(* IEC 61131-3 sources: iec-checker/test/st/good, 22 files *)

(* ---- function-declaration.st ---- *)
(* Test for declaration of Function POU. *)
FUNCTION fn1 : INT
    VAR_INPUT
        vi1 : INT;
        vi2 : DINT;
    END_VAR
    VAR_OUTPUT
        vo1 : INT;
    END_VAR
    VAR_IN_OUT
        vio1 : INT;
    END_VAR
    VAR_IN_OUT
        vio1 : INT;
    END_VAR
    VAR
        v1 : INT;
    END_VAR
    VAR_EXTERNAL
        ve1 : INT;
    END_VAR
    VAR_TEMP
        vt1 : INT;
    END_VAR

    vio1 := 42;
END_FUNCTION

(* ---- generic-types.st ---- *)
(* Extended example from Beckhoff: https://infosys.beckhoff.com/english.php?content=../content/1033/tc3_plc_intro/18014401038986379.html&id= *)
FUNCTION F_AnyBitFunc : BOOL
VAR_INPUT
  value : ANY_BIT;
END_VAR
  value := 0;
END_FUNCTION

FUNCTION F_AnyDateFunc : BOOL
VAR_INPUT
    value : ANY_DATE;
END_VAR
  value := 0;
END_FUNCTION

FUNCTION F_AnyFunc : BOOL
VAR_INPUT
    value : ANY;
END_VAR
  value := 0;
END_FUNCTION

FUNCTION F_AnyIntFunc : BOOL
VAR_INPUT
    value : ANY_INT;
END_VAR
  value := 0;
END_FUNCTION

FUNCTION F_AnyNumFunc : BOOL
VAR_INPUT
    value : ANY_NUM;
END_VAR
  value := 0;
END_FUNCTION

FUNCTION F_AnyRealFunc : BOOL
VAR_INPUT
    value : ANY_REAL;
END_VAR
  value := 0;
END_FUNCTION

FUNCTION F_AnyStringFunc : BOOL
VAR_INPUT
    value : ANY_STRING;
END_VAR
  value := 0;
END_FUNCTION

(* ---- array-use.st ---- *)
FUNCTION_BLOCK MAIN_POU

  VAR
      i:INT;
      state: INT:=0;
  END_VAR

   IF gvl.CALL_LIST_INTERMEDIATE_GO_UP[i]= TRUE THEN
      state:=100;
  END_IF

END_FUNCTION_BLOCK

(* ---- empty-body.st ---- *)
(* Allow POU that contains only {} in their bodies. *)
FUNCTION EmptyFun : BOOL
  {}
END_FUNCTION

FUNCTION_BLOCK EmptyFB
  {}
END_FUNCTION_BLOCK

PROGRAM EmptyProgram
  {}
END_PROGRAM

(* ---- function-blocks.st ---- *)
FUNCTION_BLOCK fb0
END_FUNCTION_BLOCK

FUNCTION_BLOCK fb1
  VAR_INPUT
    vi1 : DINT;
  END_VAR
  VAR_OUTPUT
    vo1 : DINT;
  END_VAR
  VAR_IN_OUT
    vio1 : DINT;
  END_VAR
  VAR
    v1 : DINT;
  END_VAR
  VAR_TEMP
    vt1 : DINT;
  END_VAR
  VAR RETAIN
    vr1 : DINT;
  END_VAR
  VAR NON_RETAIN
    vnr1 : DINT;
  END_VAR
  v1 := 42;
END_FUNCTION_BLOCK

(* ---- references.st ---- *)
FUNCTION_BLOCK fb1
  VAR_INPUT
    vi1 : DINT;
  END_VAR
  v1 := 42;
END_FUNCTION_BLOCK

PROGRAM example
  VAR
    temp : DINT;
  END_VAR

  temp ?= temp^;
  temp ?= temp^^;
  temp ?= temp^^^;
  temp ?= NULL;
  temp ?= fb1;
END_PROGRAM

(* ---- simple.st ---- *)
FUNCTION_BLOCK Example
    VAR_EXTERNAL
        global_var : INT;
    END_VAR
    global_var := 42;
END_FUNCTION_BLOCK

PROGRAM Simple
  VAR_INPUT
    x : TIME;
  END_VAR
  VAR
    temp : DINT;
    i : DINT;
    arr1: ARRAY [1..2] OF BOOL;
    unused_var AT %IW1.2 : REAL := 200.0;
    head AT %B0 : INT;
  END_VAR

  WHILE i < 10 DO
    IF i = 5 THEN
      temp := i;
      EXIT;
      i := 42;
    END_IF
    i := i + 1;
  END_WHILE

  ARR1[3] := 19;
  ARR1[2,1] := 19;
  IF x = T#100MS THEN
    %B0 := 42;
  END_IF
END_PROGRAM

(* ---- user3.st ---- *)
FUNCTION_BLOCK MAIN_POU

  VAR_INPUT
  END_VAR

  VAR_OUTPUT
  END_VAR

  VAR
      FB4_Populate_Intermediate_Call_List_call : FB4_Populate_Intermediate_Call_List;
      FB5_Trigger_FB2_Call_FIFO_call:FB5_Trigger_FB2_Call_FIFO;
      MC_power_X1 : MC_Power;
      MC_readAxisPosition_jog:MC_ReadActualPosition;
      MC_ReadStatus_jog:MC_ReadStatus;
      MC_jog:MC_Jog;
      MC_Halt_jog:MC_Halt;
      MC_Stop_jog:MC_Stop;
      MC_Reset_jog:MC_Reset;
      MC_MoveAbsolute_jog:MC_MoveAbsolute;
      mainMotor:Motor;
      ton_0 : TON;
      ton_1 : TON;
      ton_2 : TON;
      axisPosition:REAL;
      nextTargetFloor:INT;
      nextTargetPosition:REAL;
      nextIntermediateTargetPosition:REAL;
      nextIntermediateTargetFloor:INT;
      nextIntermediateTargetFloorAvailable:bool;
      lastTargetFloor:INT;
      currentFloorNumber_:INT;
      i:INT;
      state: INT:=0;
      test_READ:BOOL;
      test_FORWARD:BOOL;
  END_VAR

  // Write values to Global Variables
  gvl.state_POU_1:=state;
  gvl.QW_axisPosition:=axisPosition;

  // Read axis position all the time
  MC_readAxisPosition_jog(Axis:=X1,
      Enable:=TRUE,
      Position=>axisPosition);

  // Motor Halt
  IF mainMotor.IX_Halt THEN
      MC_jog(Axis:=X1,
          JogForward:=FALSE,
          JogBackward:=FALSE);
  END_IF

  // Main Power
  mainMotor.IX_Power:=TRUE;
  IF mainMotor.IX_Power THEN
      MC_power_X1(Axis:=X1,
          Enable:=TRUE,
          bRegulatorOn:=TRUE,
          bDriveStart:=TRUE);
  ELSE
      MC_power_X1(Axis:=X1,
          Enable:=FALSE,
          bRegulatorOn:=FALSE,
          bDriveStart:=FALSE);
  END_IF

  // STOP/RESET the motor
  MC_Stop_jog(Axis:=X1,
      Execute:=mainMotor.IX_Stop,
      Deceleration:=5);
  MC_Reset_jog(Axis:=X1,
      Execute:=mainMotor.IX_Reset);

  // Drive error ID
  gvl.jogErrorID := MC_jog.ErrorId;

  CASE state OF
      0:  // Power ON
          IF MC_power_X1.Status = TRUE THEN
              ton_0(IN:=NOT ton_0.Q,PT:=1);
              IF ton_0.Q THEN
                  state := 10;
              END_IF
          END_IF

      10:
          IF nextIntermediateTargetFloorAvailable=FALSE THEN
              FB5_Trigger_FB2_Call_FIFO_call(POP:=2);
              IF FB5_Trigger_FB2_Call_FIFO_call.done = TRUE THEN
                  state:=11;
              END_IF
          ELSE
              state:=11;
          END_IF

      11:
          IF gvl.Dout <>0 THEN
              state:=12;
          ELSE
              state:=10;
          END_IF

      12:
          gvl.targetPosition := WORD_TO_INT(gvl.Dout-1)*gvl.floor_to_floor_distance;
          nextTargetFloor := WORD_TO_INT(gvl.Dout);

          IF gvl.Dout <> 0 AND gvl.targetPosition <> gvl.QW_axisPosition THEN
              IF gvl.QW_axisPosition < gvl.targetPosition THEN
                  gvl.jogDirection:='GO_UP';
                  MC_jog(Axis:=X1,
                          JogForward:=TRUE,
                          Velocity:=gvl.velocity_high,
                          Acceleration:=gvl.acceleration_high,
                          Deceleration:=gvl.deceleration_high);
              ELSIF gvl.QW_axisPosition > gvl.targetPosition THEN
                  gvl.jogDirection:='GO_DOWN';
                  MC_jog(Axis:=X1,
                          JogBackward:=TRUE,
                          Velocity:=gvl.velocity_high,
                          Acceleration:=gvl.acceleration_high,
                          Deceleration:=gvl.deceleration_high);
              END_IF
          ELSE
              state:=10;
          END_IF

          FB4_Populate_Intermediate_Call_List_call();
          IF gvl.jogDirection='GO_UP' THEN
              // If intermediate floor calls available_GO_UP
              FOR i:=1 TO gvl.NUM_FLOOR DO
                   IF gvl.CALL_LIST_INTERMEDIATE_GO_UP[i]= TRUE AND gvl.QW_axisPosition > (i-1)*gvl.floor_to_floor_distance-200 THEN
                      MC_jog(Axis:=X1,
                          JogForward:=FALSE,
                          JogBackward:=FALSE);
                      nextIntermediateTargetFloor:=i;
                      gvl.nextIntermediateTargetPosition:=(i-1)*gvl.floor_to_floor_distance;
                      state:=100;
                  END_IF
              END_FOR
              // If NO intermediate floor calls available
              IF gvl.QW_axisPosition > gvl.targetPosition-400 THEN
                  MC_jog(Axis:=X1,
                  JogForward:=FALSE,
                  JogBackward:=FALSE);
              END_IF
              IF MC_jog.Busy=FALSE THEN
                  state:=102;
              END_IF
          END_IF

          IF gvl.jogDirection='GO_DOWN' THEN
              // If intermediate floor calls available_GO_DOWN
              FOR i:=1 TO gvl.NUM_FLOOR DO
                   IF gvl.CALL_LIST_INTERMEDIATE_GO_DOWN[i]= TRUE AND gvl.QW_axisPosition < (i-1)*gvl.floor_to_floor_distance+200 THEN
                      MC_jog(Axis:=X1,
                          JogForward:=FALSE,
                          JogBackward:=FALSE);
                      nextIntermediateTargetFloor:=i;
                      gvl.nextIntermediateTargetPosition:=(i-1)*gvl.floor_to_floor_distance;
                      state:=100;
                  END_IF
              END_FOR
              // If NO intermediate floor calls available
              IF gvl.QW_axisPosition < gvl.targetPosition+400 THEN
                  MC_jog(Axis:=X1,
                  JogForward:=FALSE,
                  JogBackward:=FALSE);
              END_IF
              IF MC_jog.Busy=FALSE THEN
                  state:=102;
              END_IF
          END_IF

      100: // If YES intermediate floor calls available
          MC_MoveAbsolute_jog(Axis:=X1,
              Execute:=TRUE,
              Position:=gvl.nextIntermediateTargetPosition,
              Velocity:=gvl.velocity_low,
              Acceleration:=gvl.acceleration_low,
              Deceleration:=gvl.deceleration_low);

          IF MC_MoveAbsolute_jog.Done THEN
              MC_MoveAbsolute_jog(Axis:=X1,
                  Execute:=FALSE);
              nextIntermediateTargetFloorAvailable:=TRUE;
              state:=400;
          END_IF;

      102: // If NO intermediate floor calls available
          MC_MoveAbsolute_jog(Axis:=X1,
              Execute:=TRUE,
              Position:=gvl.targetPosition,
              Velocity:=gvl.velocity_low,
              Acceleration:=gvl.acceleration_low,
              Deceleration:=gvl.deceleration_low);

          IF MC_MoveAbsolute_jog.Done THEN
              MC_MoveAbsolute_jog(Axis:=X1,
                  Execute:=FALSE);
              nextIntermediateTargetFloorAvailable:=FALSE;
              state:=400;
          END_IF

      400: // Door closed and all safety OK.
          currentFloorNumber_:=FC1_currentFloorNumber(axisPosition:=axisPosition);
          gvl.Din_toRemove := INT_TO_WORD(currentFloorNumber_);

          gvl.CALL_LIST[currentFloorNumber_]:=FALSE;
          gvl.CALL_LIST_INTERMEDIATE_GO_DOWN[currentFloorNumber_]:=FALSE;
          gvl.CALL_LIST_INTERMEDIATE_GO_UP[currentFloorNumber_]:=FALSE;

          FB5_Trigger_FB2_Call_FIFO_call(POP:=3);
          IF FB5_Trigger_FB2_Call_FIFO_call.done = TRUE THEN
              state:=402;
          END_IF

      402:
          IF GVL.IX_DoorClosedAndAllSafetyOk THEN
              state:=10;
          END_IF

  END_CASE

END_FUNCTION_BLOCK

(* ---- array-in-loop.st ---- *)
PROGRAM Simple

  VAR
    i : DINT;
    arr1: ARRAY [1..2] OF BOOL;
  END_VAR

  VAR
    unused_var AT %IW1.2 : REAL := 200.0;
  END_VAR

  IF ARR1[i] < 10 THEN
    i := i + 1;
  END_IF;
END_PROGRAM

(* ---- case-insensitive.st ---- *)
(* Keywords and identifiers are case-insensitive *)
Program simple
  VaR
    v01 : DiNt;
  eND_var

  v01 := 92;
  V01 := 92;
END_PROGRAM

PRoGRAM square_root
  var
    a, b, c, d : REAL;
    x1, x2 : REaL;
    nroots : InT;
  END_VAR

  d := b*b - 4.0*a;
  d := b*b - 4.0*a*c;
  IF d < 0.0
  THEN nroots := 0;
    ELSIF d = 0.0
    THEN
      nroots := 1;
      X1 := -b/(2.0*A);
      X1 := -b;
    ELSE
      nroots := 2;
      X1 := (-b + SQRT(d))/(2.0*a);
      X2 := (-b - SQRT(d))/(2.0*a);
  END_IF;

ENd_ProGRAM

(* ---- comments.st ---- *)
PROGRAM comments
	VAR
		INITIAL : BOOL := FALSE;
		X1 : INT := 10;
		Y1 : INT := 20;
    // Test
	END_VAR
  // Test1
	Y1 := Z + 1; // Test2
	O_I1 := Y1; // Test3
END_PROGRAM

(* ---- configurations.st ---- *)
(* Demo program with all possible TASK entries.
   Created with Beremiz IDE (https://beremiz.org/). *)
FUNCTION function0 : BOOL
  VAR
    LocalVar0 : DINT;
  END_VAR

  LocalVar0 := 42;
END_FUNCTION

PROGRAM program0
  VAR
    LocalVar0 : DINT;
    LocalVar1 : TOD;
  END_VAR

  LocalVar0 := 42;
END_PROGRAM

PROGRAM program1
  VAR
    LocalVar0 : DINT;
  END_VAR

  LocalVar0 := 16#42;
END_PROGRAM

CONFIGURATION config
  VAR_GLOBAL
    ConfVar0 : DINT;
    ConfVar1 : DINT;
    ConfVar2 : DINT;
  END_VAR

  RESOURCE resource1 ON PLC
    VAR_GLOBAL
      ResVar0 : DINT;
      ResVar1 : BOOL;
    END_VAR
    TASK task0(INTERVAL := T#20ms,PRIORITY := 0);
    TASK task1(SINGLE := ResVar1,PRIORITY := 0);
    TASK task2(INTERVAL := T#2h0m0s3ms,PRIORITY := 1);
    PROGRAM instance0 WITH task0 : program0;
    PROGRAM instance1 WITH task1 : program1;
    PROGRAM instance2 WITH task2 : program1;
  END_RESOURCE
END_CONFIGURATION

(* ---- control-statements.st ---- *)
(* This file contains various control statements of the ST language. *)

(* Table 72 -- №4 *)
PROGRAM square_root
  VAR
    a, b, c, d : REAL;
    x1, x2 : REAL;
    nroots : INT;
  END_VAR

  d := b*b - 4.0*a;
  d := b*b - 4.0*a*c;
  IF d < 0.0
  THEN nroots := 0;
    ELSIF d = 0.0
    THEN
      nroots := 1;
      X1 := -b/(2.0*A);
      X1 := -b;
    ELSE
      nroots := 2;
      X1 := (-b + SQRT(d))/(2.0*a);
      X2 := (-b - SQRT(d))/(2.0*a);
  END_IF;

END_PROGRAM

PROGRAM test_for
  VAR
    i, j : INT;
    flag : INT;
    counter : INT := 0;
    some_var : INT;
  END_VAR

  FOR i := 0 TO 10 DO
    FOR j := 10 TO 100 BY 2 DO
      IF flag THEN
        EXIT;
      END_IF;
      counter := counter + 1;
      IF j = 10 THEN
        CONTINUE;
      END_IF;
    END_FOR;
  END_FOR;
END_PROGRAM

PROGRAM test_switch_case
  VAR
    TW : INT;
    THUMBWHEEL : WORD;
    TW_ERROR : INT;
    some_var : INT;
  END_VAR

  TW := WORD_BCD_TO_INT(THUMBWHEEL);
  TW_ERROR:= 0;
  CASE TW OF
    1,5:     DISPLAY := OVEN_TEMP;
    2:       DISPLAY := MOTOR_SPEED;
    3:       DISPLAY := GROSS - TARE;
    4,6..10: DISPLAY := STATUS(TW-4);
  ELSE DISPLAY := 0;
       TW_ERROR:= 1;
  END_CASE;
  QW100:= INT_TO_BCD(DISPLAY);
END_PROGRAM

FUNCTION fn0 : INT
  VAR_INPUT
    INVAL : INT;
  END_VAR
  VAR_OUTPUT
    OUTVAL : INT;
  END_VAR

  OUTVAL := 0;
END_FUNCTION

PROGRAM p0
  VAR_INPUT
    vi1 : INT;
  END_VAR
  VAR_OUTPUT
    vo1 : INT;
    vo2 : INT;
  END_VAR
  VAR
    i : INT;
    x : INT;
    acc : INT;
    j : INT;
  END_VAR

  IF (vi1 = 0)
    THEN vo1 := 0;
    ELSE vo1 := vi1 - 42;
  END_IF;

  CASE vi1 OF
    1 : vo1 := 19;
    2 : vo1 := 29;
    3,4 : vo1 := 39;
    (* TODO: 3..10: vo1 := 42; *)
    ELSE vo1 := 1; vo2 := -1;
  END_CASE;

  FOR i := 1 TO 100 DO
    acc := acc * x;
  END_FOR;

  FOR i := 100 TO 0 BY -2 DO
    acc := acc * x;
  END_FOR;

  J := 1;
  WHILE J <= 100 DO
    J := J + 2;
  END_WHILE;

  J := -1;
  REPEAT
    J := J + 2;
    UNTIL J = 101
  END_REPEAT;

  (* Invocation statements *)
  acc := fn0();
  acc := fn0(19);
  acc := fn0(INVAL := 19);

END_PROGRAM

(* ---- direct-variables.st ---- *)
(* Examples of directly represented variables from ch. 6.5.5 *)
PROGRAM simple
  VAR
    v01 AT %IW215 : DINT;
    v02 AT %QB7 : DINT;
    v03 AT %MD48 : DINT;
    v04 AT %IX1 : DINT;
    v05 AT %I1 : DINT;
    v06 AT %IB2 : DINT;
    v07 AT %IW3 : DINT;
    v08 AT %ID4 : DINT;
    v09 AT %IL5 : DINT;
    v10 AT %IB0 : DINT;
    v11 AT %QX7.5 : DINT;
    v12 AT %MW1.7.9 : DINT;
    v13 AT %M* : DINT;
    v14 AT %MW10.2.4.1 : INT;
		v15 AT %MW11 : INT;
		v16 AT %MW12: INT;
  END_VAR

  v01 := 92;
END_PROGRAM

(* ---- literals.st ---- *)
(* Test lexing/parsing of literals. *)
PROGRAM program0
  VAR
    a : ULINT;
    b : BOOL;
    r : REAL;
    t : TIME;
    td : TOD;
    d : DATE;
    dtv : DATE_AND_TIME;

    (* The following identifiers are not defined as reserved keywords in the standard.
       So they could be used as a regular identifiers. *)
    T : INT;
    LT : INT;
    D : INT;
    LD : INT;

    s : STRING;
    x : BYTE;
    y : WORD;
    z : DWORD;
    w : LWORD;
  END_VAR

  (* integer *)
  a := 3;
  a := 3_000;
  a := 3_000_000;
  a := 3_00_0000;
  a := ULINT#3;
  a := ULINT#3_000;

  (* binary_integer *)
  a := 2#1;
  a := 2#010110;
  a := 2#11_011_0;
  a := ULINT#2#1;
  a := ULINT#2#1_000;

  (* octal_integer *)
  a := 8#7;
  a := 8#71_061_0;
  a := ULINT#8#7;
  a := ULINT#8#7_000;

  (* hex_integer *)
  a := 16#0;
  a := 16#10;
  a := 16#A;
  a := 16#A_B_C;
  a := ULINT#16#A;
  a := ULINT#16#A_B00;

  (* bool_literal *)
  b := 1;
  b := 0;
  b := FALSE;
  b := TRUE;
  b := BOOL#1;
  b := BOOL#0;
  b := BOOL#FALSE;
  b := BOOL#TRUE;

  (* real_lieral *)
  r := 1.0;
  r := 0.0;
  r := 3.000_300;
  r := +3.2;
  r := 3.2E1;
  r := +3.2E1;
  r := -3.2E1;
  r := -3.2E+1;
  r := -3.2E-1;
  r := REAL#2.0;
  r := REAL#-2.0;
  r := REAL#-2.0E8;
  r := REAL#-2.0E-8;

  (* time_literal *)
  t := TIME#3.0d;
  t := TIME#3d;
  t := TIME#3.0h;
  t := TIME#3.0m;
  t := TIME#3.0s;
  t := TIME#3.0ms;
  t := TIME#3.0us;
  t := TIME#3.0ns;
  t := TIME#3.0d 4.0h;
  t := TIME#3.0h3m;
  t := LTIME#3.0d;
  t := T#3.0d;
  t := LT#3.0d;
  t := TIME#3.0d;

  (* time_of_day *)
  td := TOD#03:12:20;
  td := LTOD#03:12:20;
  td := TIME_OF_DAY#03:12:20;
  td := LTIME_OF_DAY#03:12:20;
  td := LTIME_OF_DAY#03:12:20.5;

  (* date *)
  d := DATE#2020-01-30;
  d := LDATE#2020-01-30;
  d := D#2020-01-30;
  d := LD#2020-01-30;

  (* date_and_time *)
  dtv := LDT#2020-01-30-18:01:38;
  dtv := LDT#2020-01-30-18:01:38.33;
  dtv := DT#2020-01-30-18:01:38;
  dtv := DATE_AND_TIME#2020-01-30-18:01:38;
  dtv := LDATE_AND_TIME#2020-01-30-18:01:38;

  (* String literals *)
  s := "FOO";
  s := "(*FO*)O";
  s := 'BAR';
  s := STRING#"FOO";
  s := STRING#"BAR(*";
  s := STRING#'FOO';

  x := BYTE#8#01;
  y := WORD#16#1234;
  z := DWORD#12345678;
  w := LWORD#2#10100101001010101010101010101010;

END_PROGRAM
(* vim: set foldmethod=marker foldlevel=0 foldenable sw=2 tw=120 : *)

(* ---- multiple-pous.st ---- *)
FUNCTION function0 : BOOL
  VAR
    LocalVar0 : DINT;
    LocalVar0_ : DINT;
  END_VAR
  LocalVar0 := LocalVar0 / 2;
END_FUNCTION

PROGRAM program0
  VAR_ACCESS
    acc : Var1 : DINT;
    acc : Var2 : DINT;
  END_VAR
  Var1 := 19 / 0;
  Var2 := Var1 / 1;
  Var2 := Var2 / 0;
END_PROGRAM

FUNCTION function1 : BOOL
  VAR
    LocalVar0 : DINT;
    LocalVar0_ : DINT;
  END_VAR
  LocalVar0 := LocalVar0 / 2;
END_FUNCTION

(* ---- multiple-variables.st ---- *)
PROGRAM program0
  VAR_ACCESS
    dummy : va1 : DINT;
    dummy : va2 : DINT;
    dummy : va3 : DINT;
  END_VAR
  VAR_INPUT
    vi1, vi2 : DINT;
    vi3, vi4, vi5 : DINT;
    vi6 : DINT;
  END_VAR
  VAR_OUTPUT
    vo1, vo2 : DINT;
    vo3, vo4, vo5 : DINT;
    vo6 : DINT;
  END_VAR
  VAR_IN_OUT
    vio1, vio2 : DINT;
    vio3, vio4, vio5 : DINT;
    vio6 : DINT;
  END_VAR
  VAR
    v1, v2 : DINT;
    v3, v4, v5 : DINT;
    v6 : DINT;
  END_VAR
  VAR_EXTERNAL
    ve1 : DINT;
    ve2 : DINT;
    ve3 : DINT;
  END_VAR
  VAR_TEMP
    vt1 : DINT;
    vt2 : DINT;
    vt3 : DINT;
  END_VAR
  VAR
    vinc1 AT %Q* : INT;
    vinc2 AT %I* : INT;
    vinc3 AT %M* : INT;
  END_VAR
  VAR
    v1 : DINT;
    v2 AT %M* : INT;
  END_VAR

  vi1 := vi1 / 1;
END_PROGRAM

(* ---- struct-declaration.st ---- *)
TYPE example_struct :
  STRUCT
    X : DINT;
    Y : BOOL;
    Z : STRING[40];
  END_STRUCT
END_TYPE

PROGRAM Program1
  VAR
    instance AT %MW500 : example_struct;
  END_VAR

  // Write the first character of Z:
  %MW504 := 'E';
END_PROGRAM

(* ---- time-literals.st ---- *)
PROGRAM program0
  VAR
    A : INT;
    T : INT;
  END_VAR

  A := 1;
END_PROGRAM

(* ---- types.st ---- *)
(* This file contains variables with valid type definitions. *)
TYPE
  (* Character strings *)
  S : STRING;
  S1 : STRING[5];
  WS : WSTRING;
  WS1 : WSTRING[5];
  WS1 : WSTRING[25] := 'spaces_disallowed';
  C : CHAR;
  WC : WCHAR;

  (* Subrange types *)
  ANALOG_DATA : INT (-4095 .. 4095);

  (* Enum types *)
  Traffic_Light: (Red, Amber, Green);
  Painting_colors: (Red, Yellow, Blue) := Blue;

  (* Array types *)
  BITS: ARRAY [0..7] OF BOOL := [0,1,1,0,0,1,0,0];

  (* Struct types *)
  ANALOG_CHANNEL_CONFIGURATION: STRUCT
    RANGE: ANALOG_SIGNAL_RANGE;
    MIN_SCALE: INT := -4095;
    MAX_SCALE: INT := 4095;
  END_STRUCT;
  Cooler: STRUCT
    Temp: INT;
    Cooling: TOF;
  END_STRUCT;
  Com1_data: STRUCT
    head AT %B0 : INT;
    length AT %B2 : USINT := 26;
    flag1 AT %X3.0 : BOOL;
    end AT %B25 : BYTE;
  END_STRUCT;
END_TYPE

PROGRAM arr_demo
  VAR
    myAnalog_16: ARRAY [1..16] OF DINT;
    TBT1 : ARRAY [1..2, 1..3] OF INT;
    BITS: ARRAY [0..7] OF BOOL := [0,1,1,0,0,1,0,0];
  END_VAR
  myAnalog_16[0] := 3;
END_PROGRAM

(* ---- user1.st ---- *)
(* a simple ST program that call a user defined function, and executes a FOR loop *)
PROGRAM prog1

	VAR_TEMP RETAIN

		I, Z : INT ;
		INITIAL : BOOL := FALSE;
		X1 : INT := 10;
		Y1 : INT := 20;
		R1 : REAL := 3.0;
		A : BOOL := TRUE;
		DI1 : BOOL := FALSE;

		I_I1 AT %MW10.2.4.1 : INT;
		I_I2 AT %MW11 : INT;
		O_I1 AT %QW63.1 : INT;

	END_VAR

  (* currently we allow GLOBAL blocks inside PROGRAMS *)
	VAR_GLOBAL
		G1: BOOL;
	END_VAR

	IF INITIAL = FALSE THEN
		I_I2 := 100;
		INITIAL := TRUE;
	END_IF;

	Z := func1(X1, Y1); // user defined function

	A := A AND G1;

	G1 := NOT G1; // changes in each run

	Y1 := Z + 5;

	FOR I := 1 TO 3 DO
		R1 := SQRT(R1);
		X1 := I;
	END_FOR;

	Y1 := Z + 1;
	O_I1 := Y1;

END_PROGRAM

(* ---- variables-declaration.st ---- *)
PROGRAM REF_DEMO
  (* Elementary *)
  VAR
    v : INT;
    v : INT := 1;
    v : BOOL;
    v : BOOL := FALSE;
    v : REAL := 10.0;
  END_VAR

  (* Direct and partly-located *)
  VAR
    v AT %IW1.2 : REAL;
    v AT %IW1.2 : REAL := 200.0;
  END_VAR

  (* Reference variables *)
  VAR
    myRefInt: REF_TO INT;
  END_VAR

  (* Arrays *)
  VAR
    A : ARRAY[0..5] OF INT;
    A : ARRAY[0..5] OF INT := [1,2,3];
    aWStrings: ARRAY[0..1] OF WSTRING := ["1234", "5678"];
  END_VAR

  (* Empty case *)
  VAR
  END_VAR

  (* Retain / non-retain variables *)
  VAR RETAIN foo : INT; END_VAR
  VAR NON_RETAIN bar : INT; END_VAR

  myRefInt := 1;
END_PROGRAM

PROGRAM no_variables
  myRefInt := 1;
END_PROGRAM
